// TwinCAT 3 PLC project PLC
// ProgramVersion: 3.1.4024.0
// libraries:
//   Tc2_Standard, * (Beckhoff Automation GmbH)
//   Tc2_System, * (Beckhoff Automation GmbH)
//   Tc3_Module, * (Beckhoff Automation GmbH)
//   Util, * (System)
//   VisuDialogs, * (System)
//   VisuSymbols,3.5.10.0,System
// project tree:
//   DUTs/ eStati.TcTLEO, stInput.TcDUT, stOutput.TcDUT, stRawInput.TcDUT, stRawOutput.TcDUT
//   / Gestore di visualizzazione.TcVMO (not stored), GlobalTextList.TcGTLO, PlcTask.TcTTO (not stored)
//   GVLs/ GVL_IO.TcGVL, GVL_SIM.TcGVL
//   POUs/ MAIN.TcPOU
//   POUs/MSF/auxiliar/ FB_MSF.TcPOU, FB_oscillatore.TcPOU, FB_ReadInput.TcPOU, FB_WriteOutput.TcPOU
//   POUs/Simu/DUTs/ stSimu.TcDUT
//   POUs/Simu/ FB_Simulatore.TcPOU
//   VISUs/ Visualization.TcVIS
// real-time tasks:
//   TASK PlcTask: cycle T#10ms, priority 20, ADS port 350

// ---- DUTs/eStati.TcTLEO
{attribute 'qualified_only'}
{attribute 'strict'}
TYPE eStati :
(
	S0 := 0, S1, S2, S3, SE, SA
);
END_TYPE

// ---- DUTs/stInput.TcDUT
TYPE stInput :
STRUCT
	start	:	BOOL;
	stop	:	BOOL;
	emg		:	BOOL;
	ack		:	BOOL;
	FC1		:	BOOL;
	FC2		:	BOOL;	
END_STRUCT
END_TYPE

// ---- DUTs/stOutput.TcDUT
TYPE stOutput :
STRUCT
	H1		:	BOOL;
	HEmglamp	:	BOOL;
	HEmg	:	BOOL;
	M		:	BOOL;
	Libero	:	BOOL;
	Idle	:	TIME;
END_STRUCT
END_TYPE

// ---- DUTs/stRawInput.TcDUT
TYPE stRawInput :
STRUCT
	Start	:	BOOL;
	Stop	:	BOOL;
	Emg		:	BOOL;
	Ack		:	BOOL;
	FC1		:	BOOL;
	FC2		:	BOOL;
END_STRUCT
END_TYPE

// ---- DUTs/stRawOutput.TcDUT
TYPE stRawOutput :
STRUCT
	H1		:	BOOL;
	HEmg	:	BOOL;
	M		:	BOOL;
	Libero	:	BOOL;
END_STRUCT
END_TYPE

// ---- POUs/Simu/DUTs/stSimu.TcDUT
TYPE stSimu :
STRUCT
	x0	:	INT;    // posizione iniziale pacco
	x1	:	INT;	// posizione finale pacco
	x	:	INT;	// posizione del pacco sul nastro
	invis	:	BOOL;	// pacco invisibile
	sET	:	STRING;	// tempo trascorso dall'ultimo pacco
END_STRUCT
END_TYPE

// ---- GVLs/GVL_IO.TcGVL
{attribute 'qualified_only'}
VAR_GLOBAL
	// ingressi
	start: BOOL;
	stop : BOOL;
	emg  : BOOL;
	ack  : BOOL;
	fc1  : BOOL;
	fc2  : BOOL;
	
	// uscite
	H1   : BOOL;
	HEMG : BOOL;
	M    : BOOL;
	// il nastro è libero
	libero : BOOL; 	
END_VAR

// ---- GVLs/GVL_SIM.TcGVL
{attribute 'qualified_only'}
VAR_GLOBAL
	sET	:	STRING := 'ABC';
END_VAR

// ---- POUs/MAIN.TcPOU
PROGRAM MAIN
VAR
	// flag inizializzazione
	setup	:	BOOL	:= TRUE;
	
	// variabili di processo
	input	:	stInput;
    output	:	stOutput;
	
	readInput	:	FB_ReadInput();
	nastro		:	fb_msf();
	writeOutput	:	FB_WriteOutput();
	
	// simulatore
	plant	:	FB_Simulatore();
END_VAR

IF(setup) THEN
	setup := FALSE;
	GVL_IO.rawInputs.Emg := TRUE;
	GVL_IO.rawInputs.Stop := TRUE;
	GVL_IO.rawInputs.FC1 := FALSE;
	GVL_IO.rawInputs.FC2 := FALSE;
	
ELSE
// lettura ingressi fisici
	readInput(rawInput := GVL_IO.rawInputs, input := input);
	
// esecuzione MSF
    nastro(input := input, output := output);
	
// aggiornamento uscite fisiche
	writeOutput(output := output, rawoutput := GVL_IO.rawOutputs);
	
// ----------------------------
// esecuzione simulatore
	plant(plantInput := GVL_IO.rawOutputs, plantOutput := GVL_IO.rawInputs);	

// ----------------------------
END_IF

END_PROGRAM

// ---- POUs/MSF/auxiliar/FB_ReadInput.TcPOU
FUNCTION_BLOCK FB_ReadInput
VAR_INPUT
	rawInput	:	stRawInput;
END_VAR
VAR_IN_OUT
	input	:	stInput;
END_VAR
VAR
	tpStart	:	TP();
	tpAck	:	TP();
END_VAR

// temporizzatori a impulso per start e ack
	tpStart(IN := rawInput.Start, PT := T#200MS);
	tpAck(IN := rawInput.Ack, PT := T#200MS);

// aggiornamento ingressi virtuali
	input.start := tpStart.Q;
	input.stop := rawInput.Stop;
	input.ack := tpAck.Q;
	input.emg := rawInput.Emg;
	input.FC1 := rawInput.FC1;
	input.FC2 := rawInput.FC2;

END_FUNCTION_BLOCK

// ---- POUs/MSF/auxiliar/FB_MSF.TcPOU
FUNCTION_BLOCK FB_MSF
VAR_INPUT
	input 	: stInput;
END_VAR
VAR_IN_OUT
	output	: stOutput; 	
END_VAR
VAR
	// abilitazione dell’automatismo
	enable : BOOL;

	// condizioni di transizione
	tr_S0_S1 : BOOL;
	tr_S1_S2 : BOOL;
	tr_S2_S3 : BOOL;
	tr_S3_S1 : BOOL;
	tr_S3_S0 : BOOL;
	tr_SE_SA : BOOL;
	tr_SA_S0 : BOOL;
	
	// variabile di stato
	stato : eStati := eStati.S0;

	// timers
	T31   : TON();
	TA0   : TON();

	// triggers per segnalazione nastro libero
	pckin : R_TRIG();
	pckout: R_TRIG();
	
END_VAR

//    1. aggiornamento delle condizioni di abilitazione (input.stop, allarmi, etc)
	enable := input.stop AND input.emg;

//    2. aggiornamento di timers, contatori, triggers sui fronti
	T31(IN := (stato = eStati.S3 AND enable), PT := T#10S );
	TA0(IN := (stato = eStati.SA), PT := T#10S );
	pckin(clk:= input.fc1);
	pckout(clk:= input.fc2);
	
//    3. valutazione della condizione di arresto nominale
	IF NOT input.stop AND input.emg THEN
		stato := eStati.S0;
	END_IF
	
//    4. valutazione della condizione di arresto di emergenza
	IF (stato <> eStati.S0 AND NOT input.emg) THEN
		stato := eStati.SE;
	END_IF
	
//    5. aggiornamento delle condizioni di transizione di stato
	tr_S0_S1 := enable AND input.start;
	tr_S1_S2 := enable AND input.fc1 AND NOT input.fc2;
	tr_S2_S3 := enable AND input.fc2;
	tr_S3_S1 := enable AND input.fc1 AND NOT input.fc2 AND NOT T31.Q;
	tr_S3_S0 := enable AND T31.Q;
	tr_SE_SA := enable AND input.ack;
	tr_SA_S0 := enable AND TA0.Q;

//    6. switch-case della MSF
	CASE stato OF
	eStati.S0:
	    // comando uscite
		output.H1 := FALSE;
		output.HEmg := FALSE;
		output.HEmglamp := FALSE;
		//output.Libero := FALSE;
		output.M := FALSE;
		output.Idle := T#0S;
		
		// transizione di stato
		IF tr_S0_S1 THEN
			stato := eStati.S1;
		END_IF
	eStati.S1:
	    // comando uscite
		output.H1 := TRUE;
		output.HEmg := FALSE;
		output.HEmglamp := FALSE;
		//output.Libero := FALSE;
		output.M := FALSE;
		output.Idle := T#0S;
				
		// transizione di stato
		IF tr_S1_S2 THEN
			stato := eStati.S2;
		END_IF
	eStati.S2:
	    // comando uscite
		output.H1 := TRUE;
		output.HEmg := FALSE;
		output.HEmglamp := FALSE;
		//output.Libero := FALSE;
		output.M := TRUE;
		output.Idle := T#0S;
				
		// transizione di stato
		IF tr_S2_S3 THEN
			stato := eStati.S3;
		END_IF	
	eStati.S3:
	    // comando uscite
		output.H1 := TRUE;
		output.HEmg := FALSE;
		output.HEmglamp := FALSE;
		//output.Libero := FALSE;
		output.M := TRUE;
		output.Idle := T31.ET;
				
		// transizione di stato
		IF tr_S3_S1 THEN
			stato := eStati.S1;
		ELSIF tr_S3_S0 THEN
			stato := eStati.S0;
		END_IF
		
	eStati.SE:
	    // comando uscite
		output.H1 := TRUE;
		output.HEmg := TRUE;
		output.HEmglamp := FALSE;
		//output.Libero := FALSE;
		output.M := FALSE;
		output.Idle := T#0S;
				
		// transizione di stato
		IF tr_SE_SA THEN
			stato := eStati.SA;
		END_IF
		
	eStati.SA:
	    // comando uscite
		output.H1 := TRUE;
		output.HEmg := FALSE;
		output.HEmglamp := TRUE;
		output.Libero := FALSE;
		output.M := FALSE;
		output.Idle := T#0S;
				
		// transizione di stato
		IF tr_SA_S0 THEN
			stato := eStati.S0;
		END_IF
	ELSE
		stato := eStati.SE;	
	END_CASE


//    7. comando delle uscite
//	output.H1 := stato <> eStati.S0;
//	output.HEmg := (stato = eStati.SE);
//	output.HEmglamp := (stato = eStati.SA);
//	output.M := (stato = eStati.S2) OR (stato = eStati.S3);
	
	// nastro libero se (enable = true e  pckout.q) o (fc1 libero in S1);
	// nastro occupato se enable = false o fc1.rise o stato = S0
	IF (enable AND (pckout.q)) OR (stato = eStati.S1 AND NOT input.fc1) THEN
		output.libero := TRUE;
	ELSIF (NOT enable) OR pckin.Q OR stato = eStati.S0 THEN
		output.libero := FALSE;
	END_IF

END_FUNCTION_BLOCK

// ---- POUs/MSF/auxiliar/FB_WriteOutput.TcPOU
FUNCTION_BLOCK FB_WriteOutput
VAR_INPUT
	output	:	stOutput;
END_VAR
VAR_IN_OUT
	rawOutput	:	stRawOutput;
END_VAR
VAR
	lamp	:	BLINK;
END_VAR

(* 
 * Converte le uscite virtuali in uscite fisiche del PLC
 *)

	lamp(enable:=TRUE, timelow := T#250MS, timehigh := T#250MS);

	rawOutput.H1 := output.H1;
	
	IF(output.HEmglamp) THEN
		rawOutput.HEmg := lamp.OUT;		// lampeggio
//	ELSIF(output.HEmg) THEN
//		rawOutput.HEmg := output.HEmg;	// accensione fissa
//	ELSE
//		rawOutput.HEmg := FALSE;
//	END_IF
    ELSE
		rawOutput.HEmg := output.HEmg;
	END_IF
    
	rawOutput.M := output.M;
	
	rawOutput.Libero := output.Libero;

END_FUNCTION_BLOCK

// ---- POUs/Simu/FB_Simulatore.TcPOU
FUNCTION_BLOCK FB_Simulatore
VAR_INPUT
	plantInput	:	stRawOutput;
END_VAR
VAR_IN_OUT
	plantOutput	:	stRawInput;
END_VAR
VAR
	simuVar	:	stSimu;	
	tIdle	:	TON();
	rFC1	:	R_TRIG();
	fFC2	:	F_TRIG();
	busy	:	RS();
	
	// flag inizializzazione
	setup	:	BOOL	:= TRUE;
END_VAR

IF(setup) THEN 
	setup := FALSE;
	// simulatore
	simuVar.x0 := 130;
	simuVar.x1 := 470;
	simuVar.invis := TRUE;	
END_IF

rFC1(CLK := plantOutput.FC1);
fFC2(CLK := plantOutput.FC2);



// carica nuovo pacco
IF(rFC1.Q AND NOT busy.Q1) THEN
	simuVar.invis := FALSE;
	simuVar.x := simuVar.x0;
END_IF



// scarica pacco
IF(fFC2.Q) THEN
	simuVar.invis := TRUE;
	simuVar.x := simuVar.x0;
END_IF

busy(SET := rFC1.Q, RESET1 := fFC2.Q);

// timer attesa nuovo pacco
tIdle(IN := (plantInput.M AND plantInput.Libero), PT := T#20S);
simuVar.sET := TIME_TO_STRING(tIdle.ET);
//GVL_SIM.sET := TIME_TO_STRING(tIdle.ET);

// movimentazione del pacco
IF plantInput.M THEN
	// un pacco è caricato sul nastro
	IF(simuVar.invis = FALSE) THEN 	
	  IF (simuVar.x > simuVar.x0 + 10) THEN
		plantOutput.FC1 := FALSE;
	  END_IF
	  
	  IF (simuVar.x < simuVar.x1) THEN
		// sposta il pacchetto sul nastro
		simuVar.x := simuVar.x + 1;
		plantOutput.FC2 := FALSE;
	  ELSE
		plantOutput.FC2 := TRUE;
	  END_IF
	END_IF
END_IF

END_FUNCTION_BLOCK

// ---- POUs/MSF/auxiliar/FB_oscillatore.TcPOU
FUNCTION_BLOCK FB_oscillatore
VAR_INPUT
	enable	:	BOOL;
	t_high	:	TIME;
	t_low	:	TIME;
END_VAR
VAR_OUTPUT
	q		:	BOOL;
END_VAR
VAR
	t1		:	TON();
	t2		:	TON();
END_VAR

	t1(in := enable AND NOT t2.Q, pt := t_low);
	t2(in := t1.Q, pt := t_high);
	
	q := t1.Q;

END_FUNCTION_BLOCK

// ---- GlobalTextList.TcGTLO
TEXTLIST GlobalTextList
  517 = '%s'
  898 = 'Ack'
  92 = 'EMERGENZA'
  475 = 'EMG'
  431 = 'FC1'
  77 = 'FC2'
  619 = 'H1'
  229 = 'H2'
  506 = 'Libero'
  878 = 'Load'
  795 = 'M'
  902 = 'Start'
  607 = 'Stop'
  353 = 'Unload'
END_TEXTLIST

// ---- VISUs/Visualization.TcVIS
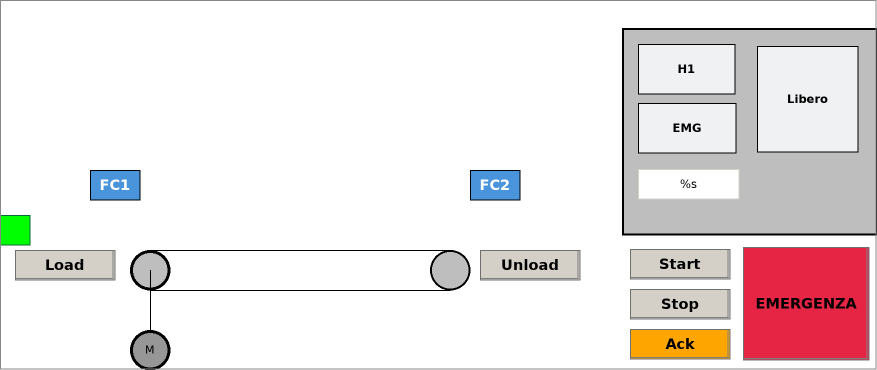
VISUALIZATION Visualization  // 877x370
    Ellipse (130,250 40x40)
    Ellipse (430,250 40x40)
    Line (150,250) (450,250)
    Line (150,290) (450,290)
    Ellipse (130,330 40x40), "M", colour toggle: GVL_IO.rawOutputs.M
    Line (150,270) (150,330)
    RoundedRectangle (622,28 255x207)
    RoundedRectangle (638,44 97x50), "H1", colour toggle: GVL_IO.rawOutputs.H1
    RoundedRectangle (638,103 98x50), "EMG", colour toggle: GVL_IO.rawOutputs.HEmg
    Textfield (638,169 101x30), "%s", text variable: MAIN.plant.simuVar.sET
    Button (630,249 100x30), "Start"
        OnMouseDown: execute { GVL_IO.rawInputs.Start := TRUE; }
        OnMouseUp: execute { GVL_IO.rawInputs.Start := FALSE; }
    Button (630,289 100x30), "Stop"
        OnMouseDown: execute { GVL_IO.rawInputs.Stop := FALSE; }
        OnMouseUp: execute { GVL_IO.rawInputs.Stop := TRUE; }
    Button (630,329 100x30), "Ack"
        OnMouseDown: execute { GVL_IO.rawInputs.Ack := TRUE; }
        OnMouseUp: execute { GVL_IO.rawInputs.Ack  := FALSE; }
    Button (743,247 126x113), "EMERGENZA"
        OnMouseDown: execute { GVL_IO.rawInputs.Emg := FALSE; }
        OnMouseUp: execute { GVL_IO.rawInputs.Emg  := TRUE; }
    RoundedRectangle (0,215 30x30), invisible if: MAIN.plant.simuVar.invis
        p3560616238: MAIN.plant.simuVar.x
    RoundedRectangle (90,170 50x30), "FC1", colour toggle: GVL_IO.rawInputs.FC1
    RoundedRectangle (470,170 50x30), "FC2", colour toggle: GVL_IO.rawInputs.FC2
    Button (15,250 100x30), "Load"
        OnMouseDown: execute { GVL_IO.rawInputs.FC1 := TRUE; }
    RoundedRectangle (757,46 101x106), "Libero", colour toggle: GVL_IO.rawOutputs.Libero
    Button (480,250 100x30), "Unload"
        OnMouseDown: execute { GVL_IO.rawInputs.FC2 := FALSE; }
END_VISUALIZATION
